// TwinCAT 3 PLC project PlcProject
// ProgramVersion: 3.1.4022.0
// libraries:
//   Tc2_Standard, * (Beckhoff Automation GmbH)
//   Tc2_System, * (Beckhoff Automation GmbH)
//   Tc3_Module, * (Beckhoff Automation GmbH)
// project tree:
//   DUTs/ ST_ComboboxEntry.TcDUT
//   / PlcTask.TcTTO
//   POUs/ MAIN.TcPOU
// real-time tasks:
//   TASK PlcTask: cycle T#10ms, priority 20, ADS port 350

CONFIGURATION PlcProject
    RESOURCE PLC ON TwinCAT3
        TASK PlcTask(INTERVAL := T#10ms, PRIORITY := 20);
        PROGRAM MAIN WITH PlcTask : MAIN;
    END_RESOURCE
END_CONFIGURATION

// ---- DUTs/ST_ComboboxEntry.TcDUT
// it is necessary that the members' names are identical to attribute names
TYPE ST_ComboboxEntry :
STRUCT
	id 	: INT;
	text 	: STRING;
	value 	: INT;
END_STRUCT
END_TYPE

// ---- POUs/MAIN.TcPOU
PROGRAM MAIN
VAR
	aComboboxEntries : ARRAY [1..9] OF ST_ComboboxEntry;
	aTexts : ARRAY [1..5] OF STRING := ['Text 1','Text 2','Text 3','Text 4','Text 5'];
	bIni: BOOL := TRUE;
	nCounter: INT;
END_VAR

// set the Combobox entries in the first cycle
IF bIni THEN
	FOR nCounter := 1 TO 5 DO
		aComboboxEntries[nCounter].id := nCounter;
		aComboboxEntries[nCounter].text := CONCAT('Array entry ', INT_TO_STRING(nCounter));
		aComboboxEntries[nCounter].value := nCounter * 10;
	END_FOR
	
	FOR nCounter := 6 TO 9 DO
		aComboboxEntries[nCounter].id := nCounter;
		aComboboxEntries[nCounter].text := CONCAT('Array entry ', INT_TO_STRING(nCounter));
		aComboboxEntries[nCounter].value := 0;
	END_FOR
	
	bIni := FALSE;
END_IF

END_PROGRAM
